// TIA Portal project "fillingTank(Timers)" (V17)
// Vorlageprojekt für das Buch mit Zielsystem S7-1200

(* hardware
DEVICE "S7-1200-Station_1"  S7-1200 Station
   slot 0: "Baugruppenträger_0"  Rack  V1.0
   slot 1: "PLC_1"  CPU 1211C DC/DC/DC  6ES7 211-1AE40-0XB0  V4.1
*)

// ===== PLC "PLC_1"  CPU 1211C DC/DC/DC =====

VAR_GLOBAL   // PLC tag table "Standard-Variablentabelle"
   "fill" AT %I0.0 : Bool;
   "discharge" AT %I0.1 : Bool;
   "factoryIORunning" AT %I0.2 : Bool;
   "fillValve" AT %Q0.0 : Bool;
   "filling" AT %Q0.1 : Bool;
   "dischargeValve" AT %Q0.2 : Bool;
   "discharging" AT %Q0.3 : Bool;
   "counter" AT %QD30 : Time;
   "temp1" AT %M0.0 : Bool;
   "Tag_1" AT %M0.1 : Bool;
   "Tag_2" AT %M0.3 : Bool;
   "Tag_3" AT %M0.5 : Bool;
   "Tag_4" AT %M0.7 : Bool;
END_VAR

DATA_BLOCK "timerValues"   // DB1
{ S7_Optimized_Access := 'TRUE' }
VERSION : 0.1
   VAR
      dataForTimer1 : Time;
      dataForTimer2 : Time;
      finalOutputT1 : Time;
      finalOutputT2 : Time;
      dataAfterSubtraction : Time;
   END_VAR
BEGIN
END_DATA_BLOCK

// folder: System blocks/Program resources

DATA_BLOCK "timer1"   // DB2
{ S7_Optimized_Access := 'TRUE' }
AUTHOR : Simatic
FAMILY : IEC
NAME : IEC_TMR
VERSION : 1.0
// stored: InstanceOfName IEC_TIMER
"IEC_TIMER"
BEGIN
END_DATA_BLOCK

DATA_BLOCK "timer3"   // DB3
{ S7_Optimized_Access := 'TRUE' }
AUTHOR : Simatic
FAMILY : IEC
NAME : IEC_TMR
VERSION : 1.0
// stored: InstanceOfName IEC_TIMER
"IEC_TIMER"
BEGIN
END_DATA_BLOCK

// folder: (top level)

FUNCTION "MHJ-PLC-Lab-Function-S71200" : Void   // FC9000, SCL
{ S7_Optimized_Access := 'TRUE' }
VERSION : 0.1
   VAR_TEMP
      rdTimeReturn : Int;
      outputTime : DTL;
      SyncVal : Byte;
      forVal : Int;
      forVal_2 : Int;
      Value : Byte;
   END_VAR
   VAR CONSTANT
      CompVal : Byte := 16#34;
      Value_01 : Byte := 16#11;
      Value_01_DW : DWord := 16#A165_D992;
      Value_02_DW : DWord := 16#58BE_4401;
   END_VAR
BEGIN

   #Value:=PEEK(area := 16#82,
        dbNumber := 0,
        byteOffset := 511);
   #Value := #Value + 1;

   POKE(area := 16#82,
        dbNumber := 0,
        byteOffset := 511,
        value := #Value);

   POKE(area:=16#81,
        dbNumber:=0,
        byteOffset:=1016,
        value:=#Value_01_DW);
   POKE(area := 16#81,
        dbNumber := 0,
        byteOffset := 1020,
        value := #Value_02_DW);

   POKE(area := 16#81,
        dbNumber := 0,
        byteOffset := 511,
        value := B#16#00);

   FOR #forVal := 0 TO 120 DO
       FOR #forVal_2:=0 TO 10 DO
           #rdTimeReturn:=RD_SYS_T(#outputTime);
           #rdTimeReturn := WR_SYS_T(#outputTime);
           #rdTimeReturn := RD_SYS_T(#outputTime);
           #rdTimeReturn := WR_SYS_T(#outputTime);
       END_FOR;
       #SyncVal:= PEEK(area := 16#81,
                      dbNumber := 0,
                      byteOffset := 511);
       IF #SyncVal = #CompVal THEN
          GOTO M_1;
       END_IF;
   END_FOR;
   RETURN;

   M_1:
   POKE(area := 16#81,
        dbNumber := 0,
        byteOffset := 511,
        value := B#16#0);
END_FUNCTION

ORGANIZATION_BLOCK "Main"   // OB1, LAD, ProgramCycle
TITLE = "Main Program Sweep (Cycle)"
{ S7_Optimized_Access := 'TRUE' }
VERSION : 0.1
   VAR_INPUT
      Initial_Call : Bool;   // Initial call of this OB
      Remanence : Bool;   // =True, if remanent data are available
   END_VAR
   VAR_TEMP   // added for the SCL form of the ladder/FBD networks
      _w1 : Bool;
   END_VAR
BEGIN

REGION Network 1: Konnektierungsbaustein für PLC-Lab
   // Im Netzwerk 1 wird der Konnektierungsbaustein für PLC-Lab aufgerufen.
   // Dieser Aufruf darf nicht entfernt werden!
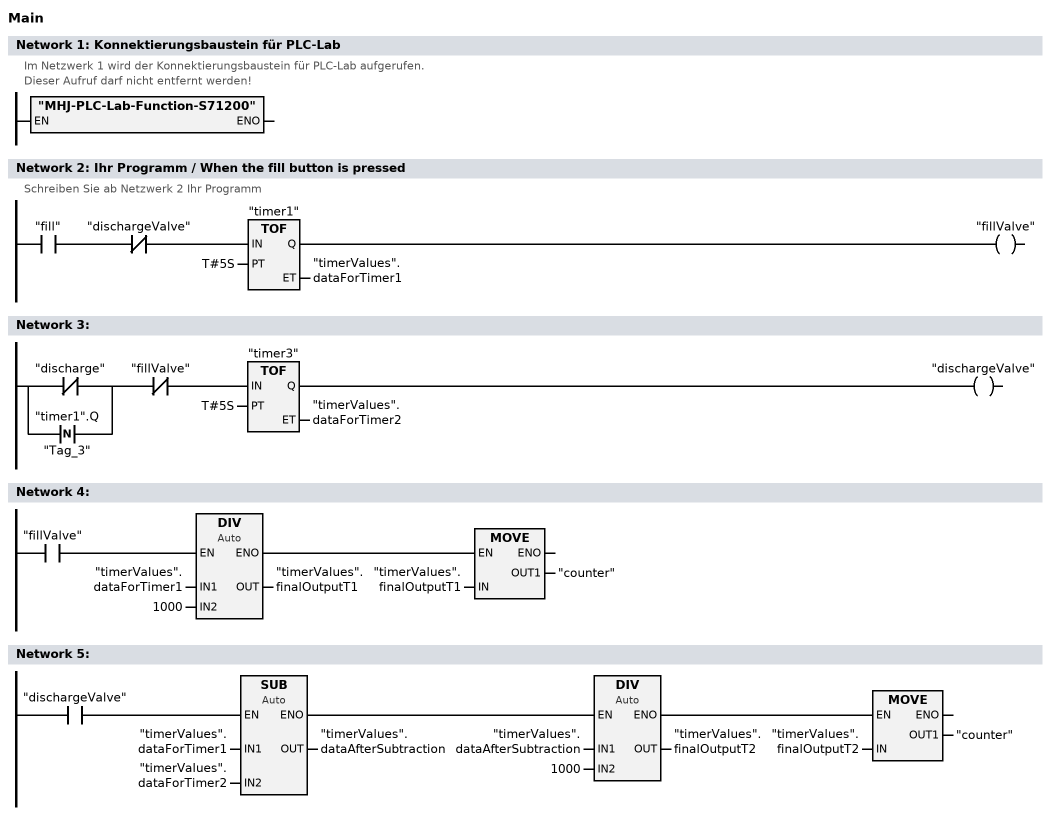
   RUNG wire#powerrail
      "MHJ-PLC-Lab-Function-S71200"()
   END_RUNG
   // the same network as SCL:
   "MHJ-PLC-Lab-Function-S71200"();
END_REGION

REGION Network 2: Ihr Programm / When the fill button is pressed
   // Schreiben Sie ab Netzwerk 2 Ihr Programm
   "timer1".TOF(IN := "fill" AND NOT "dischargeValve", PT := T#5S, ET => "timerValues".dataForTimer1);
   "fillValve" := "timer1".Q;
END_REGION

REGION Network 3
   #_w1 := NOT "timer1".Q AND "Tag_3";   // falling edge of "timer1".Q
   "Tag_3" := "timer1".Q;
   "timer3".TOF(IN := (NOT "discharge" OR #_w1) AND NOT "fillValve",
                PT := T#5S,
                ET => "timerValues".dataForTimer2);
   "dischargeValve" := "timer3".Q;
END_REGION

REGION Network 4
   RUNG wire#powerrail
      Contact( "fillValve" )
      Div(in1 := "timerValues".dataForTimer1, in2 := 1000, out => "timerValues".finalOutputT1)
      Move(in := "timerValues".finalOutputT1, out1 => "counter")
   END_RUNG
   // the same network as SCL:
   IF "fillValve" THEN
       "timerValues".finalOutputT1 := "timerValues".dataForTimer1 / 1000;
       "counter" := "timerValues".finalOutputT1;
   END_IF;
END_REGION

REGION Network 5
   RUNG wire#powerrail
      Contact( "dischargeValve" )
      Sub(in1 := "timerValues".dataForTimer1, in2 := "timerValues".dataForTimer2, out => "timerValues".dataAfterSubtraction)
      Div(in1 := "timerValues".dataAfterSubtraction, in2 := 1000, out => "timerValues".finalOutputT2)
      Move(in := "timerValues".finalOutputT2, out1 => "counter")
   END_RUNG
   // the same network as SCL:
   IF "dischargeValve" THEN
       "timerValues".dataAfterSubtraction := "timerValues".dataForTimer1 - "timerValues".dataForTimer2;
       "timerValues".finalOutputT2 := "timerValues".dataAfterSubtraction / 1000;
       "counter" := "timerValues".finalOutputT2;
   END_IF;
END_REGION
END_ORGANIZATION_BLOCK